(* PLC project OOP_Curso, Beckhoff Automation GmbH TwinCAT PLC Control 3.5.13.21 *)
(* stored: creationDateTime 2023-04-06T19:20:27.2544428, modificationDateTime 2023-04-06T19:20:27.2544428 *)

INTERFACE I_Sensor
METHOD Calibrar
END_METHOD
METHOD Descalibrar
END_METHOD
METHOD LeerValor : INT
END_METHOD
PROPERTY Consigna : REAL
END_PROPERTY
PROPERTY Temperatura : REAL
END_PROPERTY
PROPERTY Calibrado : BOOL
END_PROPERTY
END_INTERFACE

INTERFACE ITF_MyTest
METHOD METH1 : BOOL
VAR_INPUT
END_VAR
END_METHOD
METHOD METH2 : STRING
VAR_INPUT
END_VAR
END_METHOD
METHOD METH3 : REAL
VAR_INPUT
END_VAR
END_METHOD
PROPERTY Prop1 : BOOL
END_PROPERTY
PROPERTY Prop2 : REAL
END_PROPERTY
PROPERTY Prop3 : STRING
END_PROPERTY
END_INTERFACE

FUNCTION_BLOCK FB_Sensor IMPLEMENTS I_Sensor
VAR_INPUT
END_VAR
VAR_OUTPUT
END_VAR
VAR
	_Calibrar 		: BOOL;
	Valor			: INT;
	_Temperatura 	: REAL;
	_Consigna       : REAL;

END_VAR

            
          

METHOD Calibrar
                  THIS^._Calibrar := TRUE;
                
END_METHOD

METHOD Descalibrar
                  THIS^._Calibrar := FALSE;
                
END_METHOD

METHOD LeerValor : INT
                  LeerValor := Valor;
                
END_METHOD

PROPERTY Consigna : REAL
SET
VAR
END_VAR
                    THIS^._Consigna := Consigna;
                  
END_SET
END_PROPERTY

PROPERTY Temperatura : REAL
GET
VAR
END_VAR
                    Temperatura := THIS^._Temperatura;
                  
END_GET
END_PROPERTY

PROPERTY Calibrado : BOOL
GET
VAR
END_VAR
                    Calibrado := _Calibrar;
                  
END_GET
END_PROPERTY
END_FUNCTION_BLOCK

FUNCTION_BLOCK FB_TestA IMPLEMENTS ITF_MyTest
VAR_INPUT
END_VAR
VAR_OUTPUT
END_VAR
VAR
	b1: BOOL;
	r32: REAL;
	str : STRING;
END_VAR

            
          

{warning 'Agregar implementación de método'}
METHOD METH1 : BOOL
                  METH1 := TRUE;
                
END_METHOD

{warning 'Agregar implementación de método'}
METHOD METH2 : STRING
                  METH2 := 'FB_TestA';
                
END_METHOD

{warning 'Agregar implementación de método'}
METHOD METH3 : REAL
                  METH3 := 3.14;
                
END_METHOD

{warning 'Agregar implementación de propiedad'}
PROPERTY Prop1 : BOOL
GET
VAR
END_VAR
                    Prop1:= b1;
                  
END_GET
SET
VAR
END_VAR
                    b1 := Prop1;
                  
END_SET
END_PROPERTY

{warning 'Agregar implementación de propiedad'}
PROPERTY Prop2 : REAL
GET
VAR
END_VAR
                    Prop2 := r32;
                  
END_GET
SET
VAR
END_VAR
                    r32 := Prop2;
                  
END_SET
END_PROPERTY

{warning 'Agregar implementación de propiedad'}
PROPERTY Prop3 : STRING
GET
VAR
END_VAR
                    Prop3 := str;
                  
END_GET
SET
VAR
END_VAR
                    str := Prop3;
                  
END_SET
END_PROPERTY
END_FUNCTION_BLOCK

FUNCTION_BLOCK FB_TestB IMPLEMENTS ITF_MyTest
VAR_INPUT
END_VAR
VAR_OUTPUT
END_VAR
VAR
END_VAR

            
          

{warning 'Agregar implementación de método'}
METHOD METH1 : BOOL
                  
                
END_METHOD

{warning 'Agregar implementación de método'}
METHOD METH2 : STRING
                  METH2 := 'FB_TestB';
                
END_METHOD

{warning 'Agregar implementación de método'}
METHOD METH3 : REAL
                  METH3 := 8.69;
                
END_METHOD

{warning 'Agregar implementación de propiedad'}
PROPERTY Prop1 : BOOL
GET
VAR
END_VAR
                    
                  
END_GET
SET
VAR
END_VAR
                    
                  
END_SET
END_PROPERTY

{warning 'Agregar implementación de propiedad'}
PROPERTY Prop2 : REAL
GET
VAR
END_VAR
                    
                  
END_GET
SET
VAR
END_VAR
                    
                  
END_SET
END_PROPERTY

{warning 'Agregar implementación de propiedad'}
PROPERTY Prop3 : STRING
GET
VAR
END_VAR
                    
                  
END_GET
SET
VAR
END_VAR
                    
                  
END_SET
END_PROPERTY
END_FUNCTION_BLOCK

FUNCTION myFC : STRING
VAR_INPUT
	myInterface : ITF_MyTest;
END_VAR
VAR
END_VAR

            myFC := myInterface.METH2();
          
END_FUNCTION

PROGRAM _10_Interface
VAR
	//Ejemplo 1 Interface.
	Sensor 		: FB_Sensor;
	Calibrar 	: BOOL;
	Calibrado   : BOOL;
	Temperatura : REAL;
	Consigna    : REAL := 23.5;
	Valor       : INT;
	
	//Ejemplo 2 Interface.
	FB_A : FB_TestA;
	FB_B : FB_TestB;
	r32 :REAL;
	str1, str2: STRING;
	MyITF     : ITF_MyTest;
	r1, r2: REAL;
END_VAR

            // Ejemplo 1 Interface.
IF Calibrar THEN
	Sensor.Calibrar();
ELSE
	Sensor.Descalibrar();
END_IF

Calibrado := Sensor.Calibrado;
Sensor.Consigna := Consigna;

Temperatura := Sensor.Temperatura;

Valor := Sensor.LeerValor();

// Ejemplo 2 Interface.
r32:= FB_A.METH3();

str1:= myFC(FB_A);
str2:= myFC(FB_B);

MyITF := FB_A;
r1 := MyITF.METH3();
MyITF := FB_B;
r2 := MyITF.METH3();



          
END_PROGRAM
